{attribute 'GeneratedUsingTerminal: EPP7342-0002-0016'}
{attribute addProperty BoxType "EPP7342-0002-0016"}
{attribute addProperty Id "AdsAddrAT %I*.TcoAmsAddr0Chn0AT %I*USINT1Chn1AT %I*USINT1Chn2AT %I*USINT1Chn3AT %I*USINT1StateAT %I*UINT2"}
{attribute addProperty CRC "4153865593"}
{attribute addProperty Size "6"}
TYPE InfoData_F796F579 :
STRUCT
	{attribute addProperty Name "AdsAddr"}
	AdsAddr AT %I* : .TcoAmsAddr;
	{attribute addProperty Name "Chn0"}
	Chn0 AT %I* : USINT;
	{attribute addProperty Name "Chn1"}
	Chn1 AT %I* : USINT;
	{attribute addProperty Name "Chn2"}
	Chn2 AT %I* : USINT;
	{attribute addProperty Name "Chn3"}
	Chn3 AT %I* : USINT;
	{attribute addProperty Name "State"}
	State AT %I* : UINT;
END_STRUCT
END_TYPE

(* stored: Version 1.2.0.0, ProductVersion 3.1.4024.9
   DUT InfoData_F796F579: Id {12f1c242-8ca9-4521-9171-cce6bc1c1ac1} *)
